KUKA KRL program: chk_w0_wechs_ok.src

&ACCESS RV
&REL 3
&COMMENT Check Werkzeug Roboter_Bahnhof OK
DEF chk_w0_wechs_ok( )
Diag_Appl(#on,5)
;//---- Start -------
;//-- Werkzeugsignale---
;// 161--> Wkz1 Bahnhof
;// 177--> Wkz2 Bahnhof
;// 193--> Wkz3 Bahnhof
;// 209--> MPS entriegelt
;// 211--> MPS Tragplatte zusammen
;// 213--> MPS verriegelt
;//-- Werkzeugsignale---

wait for (( $in[161]) and ($in[177]) and ($in[193]) and (not $in[211]))

;//---- End -------
Diag_Appl(#Off,5)
END
